(* PLC project ClaudeUnGuided.project, Rexroth ctrlX PLC Engineering ctrlX PLC 4.6.2 *)
(* stored: creationDateTime 2026-10-09T23:34:40.7457675, modificationDateTime 2026-10-09T23:34:18.6487849 *)

PROGRAM ExampleMath
  VAR
    in1 : INT;
    in2 : INT;
    out1 : INT;
    out2 : INT;
    out3 : INT;
    out4 : INT;
    equal : BOOL;
    neq : BOOL;
    lessthan : BOOL;
    lessthanorequal : BOOL;
    GreaterThan : BOOL;
    GraterThanOrEqual : BOOL;
  END_VAR

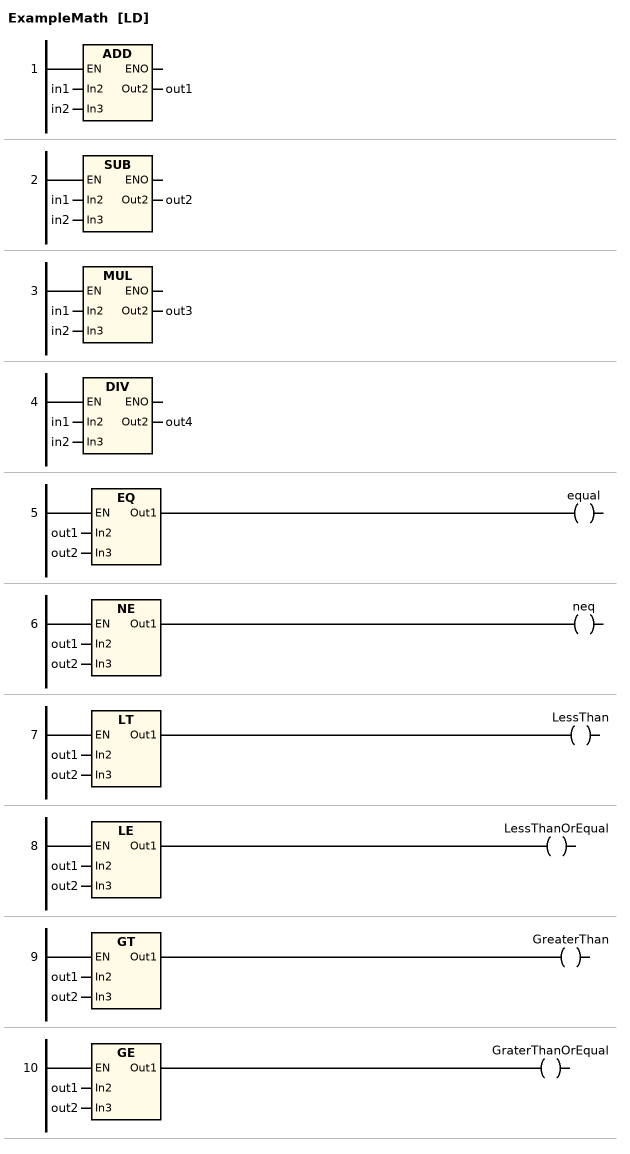
(* LD diagram, written out as Structured Text *)
(* --- network: Addition --- *)
out1 := in1 + in2;
(* --- network: Subtraction --- *)
out2 := in1 - in2;
(* --- network: Multiplication --- *)
out3 := in1 * in2;
(* --- network: Devision --- *)
out4 := in1 / in2;
(* --- network: Equate --- *)
equal := out1 = out2;
(* --- network: Not Equal --- *)
neq := out1 <> out2;
(* --- network: Less Than --- *)
LessThan := out1 < out2;
(* --- network: Less Than Or Equal TO --- *)
LessThanOrEqual := out1 <= out2;
(* --- network: Grater Than --- *)
GreaterThan := out1 > out2;

GraterThanOrEqual := out1 >= out2;
END_PROGRAM
